Fanuc KAREL source: LOCK_GROUP.kl

PROGRAM T
%NOLOCKGROUP
VAR
 v0 : INTEGER
 v1 : INTEGER
BEGIN
 LOCK_GROUP(v0, v1)
END T
